	                #sFB_RightAngledTransfer_541(iUDT_Configuration := #iUDT_Configuration."541".RightAngledTransfer,
	                                             iUDT_LowerConveyorConfiguration := #iUDT_Configuration."540".Conveyor,
	                                             iUDT_UpperConveyorConfiguration := #iUDT_Configuration."541".Conveyor,
	                                             iUDT_PECConfiguration := #iUDT_Configuration."540".PEC,
	                                             ii_DestinationA := #si_540DestinationA,
	                                             ii_DestinationB := #si_540DestinationB,
	                                             ii_DestinationC := #si_540DestinationC,
	                                             ii_DestinationD := #si_540DestinationD,
	                                             ix_HardwareOk := #ix_HardwareOk,
	                                             ix_400vOk := #ix_400vOk,
	                                             ix_24vOk := #ix_24vOk,
	                                             ix_SafetyOk := #ix_SafetyOk,
	                                             ix_AirPressureOk := #ix_AirPressureOk,
	                                             ix_SectionIsDown := #ix_SectionIsDown541,
	                                             ix_SectionIsUp := #ix_SectionIsUp541,
	                                             ix_ConveyorAAuto := #iqUDT_WorkstationCommonStatus."530".AutoON,
	                                             ix_ConveyorBAuto := #iqUDT_WorkstationCommonStatus."550".AutoON,
	                                             ix_ConveyorCAuto := #iqUDT_WorkstationCommonStatus."670".AutoON,
	                                             ix_ConveyorDAuto := FALSE,
	                                             ix_PEC := #iUDT_MotorInput540.AllSensorPortInputs.LeftSensor,
	                                             ix_ExternalReceiveRequestA := NOT #iqUDT_WorkstationStatus."530".PEC_Eos.PEC AND NOT #sx_TransferOut380 AND NOT #sx_TransferOut390,
	                                             ix_ExternalReceiveRequestB := false,
	                                             ix_ExternalReceiveRequestC := #sFB_RightAngledTransfer_671.qx_ExternalSendRequestC,
	                                             ix_ExternalReceiveRequestD := false,
	                                             ix_PECInfeedA := #iqUDT_WorkstationStatus."530".PEC_Eos.PEC,
	                                             ix_PECInfeedC := #iqUDT_WorkstationStatus."670".PEC_Eos.PEC,
	                                             qUDT_HMIRATStatus => #iqUDT_WorkstationStatus."541".RightAngledTransfer,
	                                             qUDT_HMIConveyorStatus => #iqUDT_WorkstationStatus."540".Conveyor,
	                                             qUDT_HMIPECStatus => #iqUDT_WorkstationStatus."540".PEC_Eos,
	                                             qUDT_RATStatus => #iqUDT_WorkstationCommonStatus."541",
	                                             qUDT_ConveyorStatus => #iqUDT_WorkstationCommonStatus."540",
	                                             qx_PopupControl => #qx_PopupControl541,
	                                             iqUDT_EquipmentControl := #iqUDT_EquipmentControl,
	                                             iqUDT_RATCommand := #iqUDT_WorkstationCommands."541".RightAngledTransfer,
	                                             iqUDT_ConveyorCommand := #iqUDT_WorkstationCommands."540".Conveyor,
	                                             iqUDT_RATStatistics := #iqUDT_WorkstationStatistics."541".RightAngledTransfer,
	                                             iqUDT_ConveyorStatistics := #iqUDT_WorkstationStatistics."540".Conveyor,
	                                             iqUDT_PECStatistics := #iqUDT_WorkstationStatistics."540".PEC_Eos,
	                                             iqUDT_HandShakeConveyorA := #sUDT_Handshake_530,
	                                             iqUDT_HandShakeConveyorB := #sUDT_Handshake_540,
	                                             iqUDT_HandShakeConveyorC := #sUDT_HandshakeUp_671,
	                                             iqUDT_HandShakeConveyorD := #tUDT_dummyHandshake,
	                                             iqUDT_LowerConveyorInterface := #sUDT_Interface_540,
	                                             iqUDT_UpperConveyorInterface := #sUDT_Interface_541,
	                                             iqUDT_RATPositioning := #iqUDT_RATPositioning540,
	                                             iqUDT_BladeStopEoSInterface := #tUDT_DummyBladeStop,
	                                             iqUDT_BladeStopBoSInterface := #tUDT_DummyBladeStop);

	            END_REGION

	            REGION MCO
	                #sFB_MCOConveyLinxAixController_541(iUDT_AixConfig := #iUDT_Configuration."541".MCO_M01,
	                                                    iUDT_AixInputsModule := #iUDT_MotorInput540,
	                                                    ii_PositionSetpoint := #iqUDT_RATPositioning540.Upper.EndPosition,
	                                                    ix_24vOk := #ix_24vOk,
	                                                    ix_SimulationModeActive := "DB_Memory".Simulation,
	                                                    ii_MotorPositionId := 2,
	                                                    ix_StartPositioning := #iqUDT_RATPositioning540.Upper.Start,
	                                                    ix_ResetPosition := #iqUDT_RATPositioning540.Upper.ResetPosition,
	                                                    qUDT_HMIStatus => #iqUDT_WorkstationStatus."541".MCO_M01,
	                                                    qx_Positioned => #iqUDT_RATPositioning540.Upper.Done,
	                                                    iqUDT_AixOutputsModule := #qUDT_MotorOutput540,
	                                                    iqUDT_ConveyorInterface := #sUDT_Interface_541,
	                                                    iqUDT_MCOStatistics := #iqUDT_WorkstationStatistics."541".MCO_M01);
	            END_REGION

	        END_REGION

	        REGION 550

	            REGION Displacement

	                #sFB_Displacement550(#sUDT_Interface_550);

	            END_REGION

	            REGION Tracking

	                #sFB_Tracking_550(iUDT_ConveyorCommonConfiguration := #iUDT_Configuration."550".Conveyor.Common,
	                                  iqa_TrackingData := #sa_TrackingArray_550,
	                                  iqUDT_ConveyorInterface := #sUDT_Interface_550,
	                                  iqUDT_HandshakeUp := #sUDT_Handshake_540,
	                                  iqUDT_Handshake := #sUDT_Handshake_550);
	            END_REGION

	            REGION EOS

	                #sFB_PECUpdate_550(iUDT_PECUpdateConfiguration := #iUDT_Configuration."550".PEC_EoS,
	                                   iUDT_ConveyorCommonConfiguration := #iUDT_Configuration."550".Conveyor.Common,
	                                   ix_PEC := #iUDT_MotorInput550.AllSensorPortInputs.LeftSensor,
	                                   ix_TeachingMode := FALSE,
	                                   qUDT_Status => #iqUDT_WorkstationStatus."550".PEC_EoS,
	                                   qi_GINwrite => #ti_dummy,
	                                   qx_PECFiltered => #tx_dummy,
	                                   iqa_TrackingData := #sa_TrackingArray_550,
	                                   iqUDT_ConveyorInterface := #sUDT_Interface_550,
	                                   iqUDT_UnknownGINRange := #iqUDT_UnknownGINRange,
	                                   iqUDT_FifoHeader := "DB_FIFOLostGIN".Header,
	                                   iqa_FifoData := "DB_FIFOLostGIN".Data,
	                                   iqUDT_Statistics := #iqUDT_WorkstationStatistics."550".PEC_EoS);

	            END_REGION

	            REGION Conveyor
	                #sFB_Conveyor_550(iUDT_ConveyorConfiguration := #iUDT_Configuration."550".Conveyor,
	                                  idi_PECEoSDistance := #iUDT_Configuration."550".PEC_EoS.Distance,
	                                  idi_PECBoSDistance := 0,
	                                  ii_ExternalSpeed := 0,
	                                  ix_SafetyOk := #ix_SafetyOk,
	                                  ix_24vOk := #ix_24vOk,
	                                  ix_400vOk := #ix_400vOk,
	                                  ix_HardwareOk := #ix_HardwareOk,
	                                  ix_PECEoS := #iqUDT_WorkstationStatus."550".PEC_EoS.PEC,
	                                  ix_PECBoS := TRUE,
	                                  ix_ExternalRequestHold := false,
	                                  qUDT_HMIStatus => #iqUDT_WorkstationStatus."550".Conveyor,
	                                  qUDT_Status => #iqUDT_WorkstationCommonStatus."550",
	                                  iqUDT_EquipmentControl := #iqUDT_EquipmentControl,
	                                  iqUDT_ConveyorCommand := #iqUDT_WorkstationCommands."550".Conveyor,
	                                  iqUDT_ConveyorInterface := #sUDT_Interface_550,
	                                  iqUDT_HandShakeUp := #sUDT_Handshake_540,
	                                  iqUDT_HandShake := #sUDT_Handshake_550,
	                                  iqUDT_Statistics := #iqUDT_WorkstationStatistics."550".Conveyor);
	            END_REGION

	            REGION MCO
	                #sFB_MCOConveyLinxAixController_550(iUDT_AixConfig := #iUDT_Configuration."550".MCO_M01,
	                                                    iUDT_AixInputsModule := #iUDT_MotorInput550,
	                                                    ix_24vOk := #ix_24vOk,
	                                                    ix_SimulationModeActive := "DB_Memory".Simulation,
	                                                    ii_MotorPositionId := 1,
	                                                    qUDT_HMIStatus => #iqUDT_WorkstationStatus."550".MCO_M01,
	                                                    iqUDT_AixOutputsModule := #qUDT_MotorOutput550,
	                                                    iqUDT_ConveyorInterface := #sUDT_Interface_550,
	                                                    iqUDT_MCOStatistics := #iqUDT_WorkstationStatistics."550".MCO_M01);
	            END_REGION
	        END_REGION

	        REGION 560


	            REGION Displacement

	                #sFB_Displacement560(#sUDT_Interface_560);

	            END_REGION

	            REGION Conveyor
	                #sFB_Conveyor_560(iUDT_ConveyorConfiguration := #iUDT_Configuration."560".Conveyor,
	                                  idi_PECEoSDistance := 0,
	                                  idi_PECBoSDistance := 0,
	                                  ii_ExternalSpeed := 0,
	                                  ix_SafetyOk := #ix_SafetyOk,
	                                  ix_24vOk := #ix_24vOk,
	                                  ix_400vOk := #ix_400vOk,
	                                  ix_HardwareOk := #ix_HardwareOk,
	                                  ix_PECEoS := TRUE,
	                                  ix_PECBoS := TRUE,
	                                  ix_ExternalRequestHold := false,
	                                  qUDT_HMIStatus => #iqUDT_WorkstationStatus."560".Conveyor,
	                                  qUDT_Status => #iqUDT_WorkstationCommonStatus."560",
	                                  iqUDT_EquipmentControl := #iqUDT_EquipmentControl,
	                                  iqUDT_ConveyorCommand := #iqUDT_WorkstationCommands."560".Conveyor,
	                                  iqUDT_ConveyorInterface := #sUDT_Interface_560,
	                                  iqUDT_HandShakeUp := #sUDT_Handshake_550,
	                                  iqUDT_HandShake := #sUDT_Handshake_560,
	                                  iqUDT_Statistics := #iqUDT_WorkstationStatistics."560".Conveyor);
	            END_REGION

	            REGION VFD

	                #sFB_VfdNORDPPO4_560(iUDT_VFDConfig := #iUDT_Configuration."560".VFD,
	                                     iUDT_VFDInputs := #iUDT_MotorInput560,
	                                     iUDT_MotorData := #iUDT_MotorData560,
	                                     ix_24vOk := #ix_24vOk,
	                                     ix_400vOk := #ix_400vOk,
	                                     ix_QuickStopDisable := TRUE,
	                                     ix_SimulationModeActive := "DB_Memory".Simulation,
	                                     qUDT_HMIStatus => #iqUDT_WorkstationStatus."560".VFD,
	                                     qUDT_VFDOutputs => #qUDT_MotorOutput560,
	                                     iqUDT_ConveyorInterface := #sUDT_Interface_560,
	                                     iqUDT_VFDStatistics := #iqUDT_WorkstationStatistics."560".VFD,
	                                     iqx_StartCommissioning := #iqx_StartComissioning560);

	            END_REGION

	        END_REGION

	        REGION 570

	            REGION Displacement

	                #sFB_Displacement570(#sUDT_Interface_570);

	            END_REGION

	            REGION EoS

	                #sFB_PEC_570(ix_PEC := #iUDT_MotorInput570.AllSensorPortInputs.LeftSensor,
	                             iUDT_PECConfiguration := #iUDT_Configuration."570".PEC_EoS,
	                             qUDT_HMIStatus => #iqUDT_WorkstationStatus."570".PEC_EoS,
	                             iqUDT_ConveyorInterface := #sUDT_Interface_570,
	                             iqUDT_PECStatistics := #iqUDT_WorkstationStatistics."570".PEC_EoS);

	            END_REGION

	            REGION Conveyor
	                #sFB_Conveyor_570(iUDT_ConveyorConfiguration := #iUDT_Configuration."570".Conveyor,
	                                  idi_PECEoSDistance := #iUDT_Configuration."570".PEC_EoS.Distance,
	                                  idi_PECBoSDistance := 0,
	                                  ii_ExternalSpeed := 0,
	                                  ix_SafetyOk := #ix_SafetyOk,
	                                  ix_24vOk := #ix_24vOk,
	                                  ix_400vOk := #ix_400vOk,
	                                  ix_HardwareOk := #ix_HardwareOk,
	                                  ix_PECEoS := #iqUDT_WorkstationStatus."570".PEC_EoS.PEC,
	                                  ix_PECBoS := TRUE,
	                                  ix_ExternalRequestHold := false,
	                                  qUDT_HMIStatus => #iqUDT_WorkstationStatus."570".Conveyor,
	                                  qUDT_Status => #iqUDT_WorkstationCommonStatus."570",
	                                  iqUDT_EquipmentControl := #iqUDT_EquipmentControl,
	                                  iqUDT_ConveyorCommand := #iqUDT_WorkstationCommands."570".Conveyor,
	                                  iqUDT_ConveyorInterface := #sUDT_Interface_570,
	                                  iqUDT_HandShakeUp := #sUDT_Handshake_560,
	                                  iqUDT_HandShake := #sUDT_Handshake_570,
	                                  iqUDT_Statistics := #iqUDT_WorkstationStatistics."570".Conveyor);
	            END_REGION

	            REGION MCO
	                #sFB_MCOConveyLinxAixController_570(iUDT_AixConfig := #iUDT_Configuration."570".MCO_M01,
	                                                    iUDT_AixInputsModule := #iUDT_MotorInput570,
	                                                    ix_24vOk := #ix_24vOk,
	                                                    ix_SimulationModeActive := "DB_Memory".Simulation,
	                                                    ii_MotorPositionId := 1,
	                                                    qUDT_HMIStatus => #iqUDT_WorkstationStatus."570".MCO_M01,
	                                                    iqUDT_AixOutputsModule := #qUDT_MotorOutput570,
	                                                    iqUDT_ConveyorInterface := #sUDT_Interface_570,
	                                                    iqUDT_MCOStatistics := #iqUDT_WorkstationStatistics."570".MCO_M01);
	            END_REGION
	        END_REGION

	        REGION 580

	            REGION Displacement

	                #sFB_Displacement580(#sUDT_Interface_580);

	            END_REGION

	            REGION EoS

	                #sFB_PEC_580(ix_PEC := #iUDT_MotorInput570.AllSensorPortInputs.RightSensor,
	                             iUDT_PECConfiguration := #iUDT_Configuration."580".PEC_EoS,
	                             qUDT_HMIStatus => #iqUDT_WorkstationStatus."580".PEC_EoS,
	                             iqUDT_ConveyorInterface := #sUDT_Interface_580,
	                             iqUDT_PECStatistics := #iqUDT_WorkstationStatistics."580".PEC_EoS);

	            END_REGION

	            REGION Conveyor
	                #iqUDT_HandshakeDownstream580.RTR := #iqUDT_HandshakeDownstream580.RTR OR #iqUDT_WorkstationStatus."580".PEC_EoS.PEC;
	                #sFB_Conveyor_580(iUDT_ConveyorConfiguration := #iUDT_Configuration."580".Conveyor,
	                                  idi_PECEoSDistance := #iUDT_Configuration."580".PEC_EoS.Distance,
	                                  idi_PECBoSDistance := 0,
	                                  ii_ExternalSpeed := 0,
	                                  ix_SafetyOk := #ix_SafetyOk,
	                                  ix_24vOk := #ix_24vOk,
	                                  ix_400vOk := #ix_400vOk,
	                                  ix_HardwareOk := #ix_HardwareOk,
	                                  ix_PECEoS := #iqUDT_WorkstationStatus."580".PEC_EoS.PEC,
	                                  ix_PECBoS := TRUE,
	                                  ix_ExternalRequestHold := false,
	                                  qUDT_HMIStatus => #iqUDT_WorkstationStatus."580".Conveyor,
	                                  qUDT_Status => #iqUDT_WorkstationCommonStatus."580",
	                                  iqUDT_EquipmentControl := #iqUDT_EquipmentControl,
	                                  iqUDT_ConveyorCommand := #iqUDT_WorkstationCommands."580".Conveyor,
	                                  iqUDT_ConveyorInterface := #sUDT_Interface_580,
	                                  iqUDT_HandShakeUp := #sUDT_Handshake_570,
	                                  iqUDT_HandShake := #iqUDT_HandshakeDownstream580,
	                                  iqUDT_Statistics := #iqUDT_WorkstationStatistics."580".Conveyor);
	            END_REGION
	            REGION MCO
	                #sFB_MCOConveyLinxAixController_580(iUDT_AixConfig := #iUDT_Configuration."580".MCO_M01,
	                                                    iUDT_AixInputsModule := #iUDT_MotorInput570,
	                                                    ix_24vOk := #ix_24vOk,
	                                                    ix_SimulationModeActive := "DB_Memory".Simulation,
	                                                    ii_MotorPositionId := 2,
	                                                    qUDT_HMIStatus => #iqUDT_WorkstationStatus."580".MCO_M01,
	                                                    iqUDT_AixOutputsModule := #qUDT_MotorOutput570,
	                                                    iqUDT_ConveyorInterface := #sUDT_Interface_580,
	                                                    iqUDT_MCOStatistics := #iqUDT_WorkstationStatistics."580".MCO_M01);
	            END_REGION
	        END_REGION
	    END_REGION
	END_IF;


END_FUNCTION_BLOCK

FUNCTION_BLOCK "FB_NerakLift"
{ S7_Optimized_Access := 'TRUE' }
VERSION : 0.1
// ATTRIBUTES
// AUTO_NUMBER = True
// BLOCK_NUMBER = 250
// END_ATTRIBUTES
   VAR_INPUT
      iUDT_Configuration { ExternalAccessible := 'False'; ExternalVisible := 'False'; ExternalWritable := 'False'} : "UDT_NerakLiftConfiguration";   // Configuration structure
      idi_PECEoSDistance { ExternalAccessible := 'False'; ExternalVisible := 'False'; ExternalWritable := 'False'} : DInt;   // PEC distance from the end of lift
      ix_SafetyOK { ExternalAccessible := 'False'; ExternalVisible := 'False'; ExternalWritable := 'False'} : Bool;   // TRUE when safety is ok
      ix_24VOk { ExternalAccessible := 'False'; ExternalVisible := 'False'; ExternalWritable := 'False'} : Bool;   // TRUE when 24V supply is ok
      ix_400VOk { ExternalAccessible := 'False'; ExternalVisible := 'False'; ExternalWritable := 'False'} : Bool;   // TRUE when 400V supply is ok
      ix_HardwareOk { ExternalAccessible := 'False'; ExternalVisible := 'False'; ExternalWritable := 'False'} : Bool;   // TRUE when hardware is ok
      iudt_IOIn { ExternalAccessible := 'False'; ExternalVisible := 'False'; ExternalWritable := 'False'} : "UDT_NerakLiftPI";   // Structure of inputs from IO Panel
   END_VAR

   VAR_OUTPUT
      qUDT_HMIStatus { ExternalAccessible := 'False'; ExternalVisible := 'False'; ExternalWritable := 'False'} : "UDT_NerakLiftStatus";   // HMI status structure
      qudt_IOOut { ExternalAccessible := 'False'; ExternalVisible := 'False'; ExternalWritable := 'False'} : "UDT_NerakLiftPO";   // Structure of outputs from IO Panel
      qx_Fault { ExternalAccessible := 'False'; ExternalVisible := 'False'; ExternalWritable := 'False'} : Bool;   // Fault active
      qx_Ready { ExternalAccessible := 'False'; ExternalVisible := 'False'; ExternalWritable := 'False'} : Bool;   // Machine ready
      qx_ExternalDieback { ExternalAccessible := 'False'; ExternalVisible := 'False'; ExternalWritable := 'False'} : Bool;   // Send external dieback to downstream conveyor
   END_VAR

   VAR_IN_OUT
      iqUDT_CommonStatus : "UDT_CommonStatus";   // Common status structure
      iqUDT_EquipmentControl : "UDT_EquipmentControl";   // Equipment control structure
      iqUDT_HandshakeUp : "UDT_ConveyorHandshake";   // Upstream handshake structure
      iqUDT_Handshake : "UDT_ConveyorHandshake";   // Downstream handshake structure
      iqUDT_Interface : "UDT_ConveyorInterface";   // Interface structure
      iqUDT_ConveyorCommand : "UDT_ConveyorCommand";   // HMI commands structure
      iqUDT_Statistics : "UDT_NerakLiftStatistics";   // Statistics structure
   END_VAR

   VAR
      sUDT_HMIStatus { ExternalAccessible := 'False'; ExternalVisible := 'False'; ExternalWritable := 'False'; S7_SetPoint := 'False'} : "UDT_NerakLiftStatus";   // HMI status structure
      sUDT_ConveyorConfiguration { ExternalAccessible := 'False'; ExternalVisible := 'False'; ExternalWritable := 'False'; S7_SetPoint := 'False'} : "UDT_ConveyorConfiguration" := (((), 0), (), (), (), 0, 200, (), (), FALSE);   // Conveyor configuration structure
      sFB_ConveyorControl { ExternalAccessible := 'False'; ExternalVisible := 'False'; ExternalWritable := 'False'; S7_SetPoint := 'False'} : "FB_Conveyor";   // Conveyor instance
      sFB_TimerOnOffDelay_B2Treshold { ExternalAccessible := 'False'; ExternalVisible := 'False'; ExternalWritable := 'False'; S7_SetPoint := 'False'} : "FB_TimerOnOffDelay";   // B2 on off delay
      sFB_TimerOnOffDelay_B3Treshold { ExternalAccessible := 'False'; ExternalVisible := 'False'; ExternalWritable := 'False'; S7_SetPoint := 'False'} : "FB_TimerOnOffDelay";   // B3 on off delay
      sFB_TimerOnOffDelay_B4Treshold { ExternalAccessible := 'False'; ExternalVisible := 'False'; ExternalWritable := 'False'; S7_SetPoint := 'False'} : "FB_TimerOnOffDelay";   // B4 on off delay
      sFB_TimerOnOffDelay_B5Treshold { ExternalAccessible := 'False'; ExternalVisible := 'False'; ExternalWritable := 'False'; S7_SetPoint := 'False'} : "FB_TimerOnOffDelay";   // B5 on off delay
      sFB_TimerOnOffDelay_B10Treshold { ExternalAccessible := 'False'; ExternalVisible := 'False'; ExternalWritable := 'False'; S7_SetPoint := 'False'} : "FB_TimerOnOffDelay";   // B10 on off delay
      sFB_TimerOnOffDelay_B11Treshold { ExternalAccessible := 'False'; ExternalVisible := 'False'; ExternalWritable := 'False'; S7_SetPoint := 'False'} : "FB_TimerOnOffDelay";   // B11 on off delay
      sR_TRIG_ProductFellDown {InstructionName := 'R_TRIG'; LibVersion := '1.0'; ExternalAccessible := 'False'; ExternalVisible := 'False'; ExternalWritable := 'False'; S7_SetPoint := 'False'} : R_TRIG;   // R_TRIG Product fell down for statistics
      sR_TRIG_CollisionDetected {InstructionName := 'R_TRIG'; LibVersion := '1.0'; ExternalAccessible := 'False'; ExternalVisible := 'False'; ExternalWritable := 'False'; S7_SetPoint := 'False'} : R_TRIG;   // R_TRIG collision detected for statistics
      sx_B2Filtered { ExternalAccessible := 'False'; ExternalVisible := 'False'; ExternalWritable := 'False'} : Bool;   // B2 sensor filtered
      sx_B3Filtered { ExternalAccessible := 'False'; ExternalVisible := 'False'; ExternalWritable := 'False'} : Bool;   // Cumulative B3 sensors filtered
      sx_B4Filtered { ExternalAccessible := 'False'; ExternalVisible := 'False'; ExternalWritable := 'False'} : Bool;   // B4 sensor filtered
      sx_B5Filtered { ExternalAccessible := 'False'; ExternalVisible := 'False'; ExternalWritable := 'False'} : Bool;   // B5 sensor filtered
      sx_B10Filtered { ExternalAccessible := 'False'; ExternalVisible := 'False'; ExternalWritable := 'False'} : Bool;   // B10 sensor filtered
      sx_B11Filtered { ExternalAccessible := 'False'; ExternalVisible := 'False'; ExternalWritable := 'False'} : Bool;   // B11 sensor filtered
   END_VAR

   VAR_TEMP
      tUDT_Statistics : "UDT_ConveyorStatistics";   // Temporary conveyor statistics structure
      tUDT_ConveyorHMIStatus : "UDT_ConveyorStatus";   // Temporary conveyor status structure
      tx_ExternalDieback : Bool;   // Upstream dieback control
      tx_Hold : Bool;   // Hold bit
      tx_GlobalResetMemory : Bool;   // Memory for global reset
   END_VAR


BEGIN
	(*
	----------------------------------------------------------------------------------------

	Version history:
	Date        | Version   | Author        | Remark
	----------------------------------------------------------------------------------------
	20/02/2024  | 1.0       | K.Pokorski    | First release TIA 17
	28/03/2024  | 1.1       | K. Pokorski   | Modifications after lift test
	16/08/2024  | 2.0       | J.Majer       | Block Interface IO changed to UDT type
	*)

	REGION 1 - Edge detection

	    #sR_TRIG_ProductFellDown(CLK := #sUDT_HMIStatus.Specific.ProductFellDown);

	    #sR_TRIG_CollisionDetected(CLK := #sUDT_HMIStatus.Specific.CollisionDetected);

	END_REGION

	REGION 2 - Filtering

	    #sFB_TimerOnOffDelay_B2Treshold(iudi_OnDelayTime := #iUDT_Configuration.CollisionSensorDelayOn,
	                                    iudi_OffDelayTime := #iUDT_Configuration.CollisionSensorDelayOff,
	                                    ix_SignalToDelay := #iudt_IOIn.ix_B2_CollisionControl,
	                                    qx_DelayedSignal => #sx_B2Filtered);

	    #sFB_TimerOnOffDelay_B3Treshold(iudi_OnDelayTime := #iUDT_Configuration.FallingThroughSensorDelayOn,
	                                    iudi_OffDelayTime := #iUDT_Configuration.FallingThroughSensorDelayOff,
	                                    ix_SignalToDelay := #iudt_IOIn."ix_B3.1FallingThrought" AND #iudt_IOIn."ix_B3.2FallingThrought" AND #iudt_IOIn."ix_B3.3FallingThrought",
	                                    qx_DelayedSignal => #sx_B3Filtered);

	    #sFB_TimerOnOffDelay_B4Treshold(iudi_OnDelayTime := #iUDT_Configuration.TailbackControlFrontSensorDelayOn,
	                                    iudi_OffDelayTime := #iUDT_Configuration.TailbackControlFrontSensorDelayOff,
	                                    ix_SignalToDelay := #iudt_IOIn.ix_B4TailbackControlFront,
	                                    qx_DelayedSignal => #sx_B4Filtered);

	    #sFB_TimerOnOffDelay_B5Treshold(iudi_OnDelayTime := #iUDT_Configuration.TailbackControlRearSensorDelayOn,
	                                    iudi_OffDelayTime := #iUDT_Configuration.TailbackControlRearSensorDelayOff,
	                                    ix_SignalToDelay := #iudt_IOIn.ix_B5TailbackControlBack,
	                                    qx_DelayedSignal => #sx_B5Filtered);

	    #sFB_TimerOnOffDelay_B10Treshold(iudi_OnDelayTime := #iUDT_Configuration.PlatformPositionSensorDelayOn,
	                                     iudi_OffDelayTime := #iUDT_Configuration.PlatformPositionSensorDelayOff,
	                                     ix_SignalToDelay := #iudt_IOIn.ix_B10_PlatforninPosition,
	                                     qx_DelayedSignal => #sx_B10Filtered);

	    #sFB_TimerOnOffDelay_B11Treshold(iudi_OnDelayTime := #iUDT_Configuration.CollisionSensorDelayOn,
	                                     iudi_OffDelayTime := #iUDT_Configuration.CollisionSensorDelayOff,
	                                     ix_SignalToDelay := #iudt_IOIn.ix_B11ColisionControl,
	                                     qx_DelayedSignal => #sx_B11Filtered);

	END_REGION

	REGION 3 - Errors

	    IF #iqUDT_EquipmentControl.Command.Reset OR #iudt_IOIn.ix_FaultReset
	    THEN
	        #sUDT_HMIStatus.Specific.CollisionDetected := FALSE;
	        #sUDT_HMIStatus.Specific.ProductFellDown := FALSE;
	    END_IF;

	    IF NOT #sx_B2Filtered AND #sx_B11Filtered AND #iUDT_Configuration.Mode = 1
	        OR NOT #sx_B2Filtered AND #iUDT_Configuration.Mode = 2
	    THEN
	        #sUDT_HMIStatus.Specific.CollisionDetected := TRUE;
	    END_IF;

	    IF NOT #sx_B3Filtered
	    THEN
	        #sUDT_HMIStatus.Specific.ProductFellDown := TRUE;
	    END_IF;

	    IF #sUDT_HMIStatus.Specific.CollisionDetected
	        OR #sUDT_HMIStatus.Specific.ProductFellDown THEN
	        #iqUDT_Interface.InternalErrorPEC := TRUE;
	    END_IF;

	END_REGION

	REGION 4 - Conveyor control

	    REGION 4.1 - Conveyor configuration

	        #sUDT_ConveyorConfiguration.Common.Length := #iUDT_Configuration.Length;
	        #sUDT_ConveyorConfiguration.Forward_Direction.EnergySaveLenght := #iUDT_Configuration.EnergySaveLength;
	        #sUDT_ConveyorConfiguration.Forward_Direction.PEC_EoSDistanceOffset := #iUDT_Configuration.PEC_EoSDistanceOffset;
	        #sUDT_ConveyorConfiguration.Forward_Direction.FirstConveyorToStart := #iUDT_Configuration.FirstConveyorToStart;
	        #sUDT_ConveyorConfiguration.CascadeTimeOnDelay := #iUDT_Configuration.CascadeTimeOnDelay;
	        #sUDT_ConveyorConfiguration.SpeedSetpointNominal := #iUDT_Configuration.SpeedSetpointNominal;
	        #sUDT_ConveyorConfiguration.Energy := #iUDT_Configuration.Energy;

	    END_REGION

	    REGION 4.2 - Tailback control

	        #tx_Hold := NOT #sx_B4Filtered AND NOT #sx_B5Filtered;

	    END_REGION

	    REGION 4.3 - Conveyor block call

	        #tx_GlobalResetMemory := #iqUDT_EquipmentControl.Command.Reset;
	        #iqUDT_EquipmentControl.Command.Reset := #iqUDT_EquipmentControl.Command.Reset OR #iudt_IOIn.ix_FaultReset;

	        #iqUDT_ConveyorCommand.ManualMode := #iudt_IOIn.ix_ManualMode;
	        #iqUDT_ConveyorCommand.ManualStartStop := FALSE;
	        #iqUDT_ConveyorCommand.ManualJog := #iudt_IOIn.ix_ManualUp OR #iudt_IOIn.ix_ManualDown;

	        #iqUDT_ConveyorCommand.Reverse :=
	        (#iUDT_Configuration.Mode = 1 AND #iudt_IOIn.ix_ManualUp)
	        OR (#iUDT_Configuration.Mode = 2 AND #iudt_IOIn.ix_ManualDown);

	        #sFB_ConveyorControl(iUDT_ConveyorConfiguration := #sUDT_ConveyorConfiguration,
	                             idi_PECEoSDistance := #idi_PECEoSDistance,
	                             idi_PECBoSDistance := 0,
	                             ii_ExternalSpeed := 0,
	                             ix_SafetyOk := #ix_SafetyOK,
	                             ix_24vOk := #ix_24VOk,
	                             ix_400vOk := #ix_400VOk,
	                             ix_HardwareOk := #ix_HardwareOk,
	                             ix_PECEoS := #sx_B5Filtered,
	                             ix_PECBoS := TRUE,
	                             ix_ReverseDirection := FALSE,
	                             ix_ExternalRequestDieBack := FALSE,
	                             ix_ExternalRequestHold := #tx_Hold,
	                             ix_ResetEnergySave := FALSE,
	                             qUDT_HMIStatus => #tUDT_ConveyorHMIStatus,
	                             qUDT_Status => #iqUDT_CommonStatus,
	                             iqUDT_EquipmentControl := #iqUDT_EquipmentControl,
	                             iqUDT_ConveyorCommand := #iqUDT_ConveyorCommand,
	                             iqUDT_ConveyorInterface := #iqUDT_Interface,
	                             iqUDT_HandShakeUp := #iqUDT_HandshakeUp,
	                             iqUDT_HandShake := #iqUDT_Handshake,
	                             iqUDT_Statistics := #tUDT_Statistics);

	        IF #iqUDT_CommonStatus.ManualRun
	            AND #iqUDT_Interface.SpeedSetpoint > 200
	        THEN
	            #iqUDT_Interface.SpeedSetpoint := 200;
	        END_IF;

	        #iqUDT_EquipmentControl.Command.Reset := #tx_GlobalResetMemory;
	        #tx_ExternalDieback := TRUE;
	        IF #sx_B10Filtered THEN
	            #tx_ExternalDieback := false;
	        END_IF;

	    END_REGION

	END_REGION

	REGION 5 - Status

	    #sUDT_HMIStatus.Status := #tUDT_ConveyorHMIStatus.Status;
	    #qUDT_HMIStatus := #sUDT_HMIStatus;

	END_REGION

	REGION 6 - Statistics

	    REGION 6.1 - Conveyor statistics mapping

	        #iqUDT_Statistics.EnergySave := #tUDT_Statistics.EnergySave;
	        #iqUDT_Statistics.ConveyorStop := #tUDT_Statistics.ConveyorStop;
	        #iqUDT_Statistics.ConveyorDown := #tUDT_Statistics.ConveyorDown;
	        #iqUDT_Statistics.ConveyorUp := #tUDT_Statistics.ConveyorUp;

	    END_REGION

	    REGION 6.2 - Collision detected time

	        IF #sUDT_HMIStatus.Specific.CollisionDetected OR #iqUDT_EquipmentControl.Command.ResetData  // Reset statistics
	        THEN

	            "FC_Statistics"(ix_Reset := #iqUDT_EquipmentControl.Command.ResetData,          // Reset statistics input
	                            ix_Activate := #sUDT_HMIStatus.Specific.CollisionDetected,         // Activate statistics functions input
	                            ix_RTrigActivate := #sR_TRIG_CollisionDetected.Q,                       // Statistics active trigger
	                            iqUDT_Statistics := #iqUDT_Statistics.CollisionDetected);               // Statistics values output

	        END_IF;

	    END_REGION

	    REGION 6.3 - Collision detected time

	        IF #sUDT_HMIStatus.Specific.ProductFellDown OR #iqUDT_EquipmentControl.Command.ResetData  // Reset statistics
	        THEN

	            "FC_Statistics"(ix_Reset := #iqUDT_EquipmentControl.Command.ResetData,          // Reset statistics input
	                            ix_Activate := #sUDT_HMIStatus.Specific.ProductFellDown,         // Activate statistics functions input
	                            ix_RTrigActivate := #sR_TRIG_ProductFellDown.Q,                       // Statistics active trigger
	                            iqUDT_Statistics := #iqUDT_Statistics.ProductFellDown);               // Statistics values output

	        END_IF;

	    END_REGION

	END_REGION

	REGION 7 - Outputs

	    #qx_Fault := #iqUDT_CommonStatus.Error;
	    #qx_Ready := NOT #iqUDT_CommonStatus.Error;
	    #qx_ExternalDieback := #tx_ExternalDieback;

	END_REGION
END_FUNCTION_BLOCK

FUNCTION_BLOCK "FB_TGWLift"
{ S7_Optimized_Access := 'TRUE' }
VERSION : 0.1
// ATTRIBUTES
// AUTO_NUMBER = True
// BLOCK_NUMBER = 272
// END_ATTRIBUTES
   VAR_INPUT
      iUDT_TGWLiftConfiguration { ExternalAccessible := 'False'; ExternalVisible := 'False'; ExternalWritable := 'False'} : "UDT_TGWLiftConfiguration";   // Lift configuration structure
      iUDT_010MotorInput { ExternalAccessible := 'False'; ExternalVisible := 'False'; ExternalWritable := 'False'} : "UDT_VfdSEWSpeedPI";   // 010 SEW inputs structure
      iUDT_020MotorInput { ExternalAccessible := 'False'; ExternalVisible := 'False'; ExternalWritable := 'False'} : "UDT_VfdSEWPositioningPI";   // 020 SEW Positioning structure
      is_ET200spPNDeviceName { ExternalAccessible := 'False'; ExternalVisible := 'False'; ExternalWritable := 'False'} : String;   // Name of ET200
      ix_010EoS { ExternalAccessible := 'False'; ExternalVisible := 'False'; ExternalWritable := 'False'} : Bool;   // End of the section - Lift conveyor
      ix_010BoS { ExternalAccessible := 'False'; ExternalVisible := 'False'; ExternalWritable := 'False'} : Bool;   // Begining of the section - Lift conveyor
      ix_010PECMiddle { ExternalAccessible := 'False'; ExternalVisible := 'False'; ExternalWritable := 'False'} : Bool;   // Middle of the section - Lift conveyor
      ix_010PECGapBegin { ExternalAccessible := 'False'; ExternalVisible := 'False'; ExternalWritable := 'False'} : Bool;   // Gap Check Beginning
      ix_010PECGapEnd { ExternalAccessible := 'False'; ExternalVisible := 'False'; ExternalWritable := 'False'} : Bool;   // Gap Check End
      iUDT_LiftPI { ExternalAccessible := 'False'; ExternalVisible := 'False'; ExternalWritable := 'False'} : "UDT_TGWLiftPI";   // Reading inputs from the input card
      ix_24vOk { ExternalAccessible := 'False'; ExternalVisible := 'False'; ExternalWritable := 'False'} : Bool;   // TRUE when 24VDC is healthy
      ix_400vOk { ExternalAccessible := 'False'; ExternalVisible := 'False'; ExternalWritable := 'False'} : Bool;   // TRUE when 400VAC is healthy
      ix_SafetyOk { ExternalAccessible := 'False'; ExternalVisible := 'False'; ExternalWritable := 'False'} : Bool;   // TRUE when safety is ok
      ix_HardwareOk { ExternalAccessible := 'False'; ExternalVisible := 'False'; ExternalWritable := 'False'} : Bool;   // TRUE when hardware is ok
      ix_MaintSupport1 { ExternalAccessible := 'False'; ExternalVisible := 'False'; ExternalWritable := 'False'} : Bool;   // Lift supporting maintenance platform 1 retracted
      ix_MaintSupport2 { ExternalAccessible := 'False'; ExternalVisible := 'False'; ExternalWritable := 'False'} : Bool;   // Lift supporting maintenance platform 2 retracted
      ix_KeySwitchStop { ExternalAccessible := 'False'; ExternalVisible := 'False'; ExternalWritable := 'False'} : Bool;   // Key switch stop
      ix_LimitSwitchUp { ExternalAccessible := 'False'; ExternalVisible := 'False'; ExternalWritable := 'False'} : Bool;   // Limit switch up
      ix_LimitSwitchDown { ExternalAccessible := 'False'; ExternalVisible := 'False'; ExternalWritable := 'False'} : Bool;   // Limit switch down
   END_VAR

   VAR_OUTPUT
      qUDT_010MotorOutput { ExternalAccessible := 'False'; ExternalVisible := 'False'; ExternalWritable := 'False'} : "UDT_VfdSEWSpeedPO";   // 010 SEW outputs structure
      qUDT_020MotorOutput { ExternalAccessible := 'False'; ExternalVisible := 'False'; ExternalWritable := 'False'} : "UDT_VfdSEWPositioningPO";   // 020 SEW positioning outputs structure
      qUDT_LiftPO { ExternalAccessible := 'False'; ExternalVisible := 'False'; ExternalWritable := 'False'} : "UDT_TGWLiftPO";   // writing outputs to the output card
   END_VAR

   VAR_IN_OUT
      iqUDT_EquipmentControl : "UDT_EquipmentControl";   // Equipment control structure
      iqUDT_TGWLiftHMICommands : "UDT_TGWLiftHmiCommands";   // HMI commands structure for lift
      iqUDT_TGWLiftCommonStatus : "UDT_TGWLiftCommonStatus";   // Common status structure for 010 conveyor
      iqUDT_TGWLiftStatus : "UDT_TGWLiftStatus";   // Status TGW Lift structure
      iqUDT_TGWLiftStatistics : "UDT_TGWLiftStatistics";   // Statistics TGW Lift structure
      iqUDT_InfeedFullDownHMICommands : "UDT_ConveyorCommand";   // HMI commands structure for lower infeed conveyor
      iqUDT_OutfeedEmptyDownHMICommands : "UDT_ConveyorCommand";   // HMI commands structure for lower outfeed conveyor
      iqUDT_InfeedEmptyUpHMICommands : "UDT_ConveyorCommand";   // HMI commands structure for upper infeed conveyor
      iqUDT_OutfeedFullUpHMICommands : "UDT_ConveyorCommand";   // HMI commands structure for upper outfeed conveyor
      iqUDT_InfeedFullDownCommonStatus : "UDT_CommonStatus";   // Common status structure for full infeed conveyor
      iqUDT_OutfeedEmptyDownCommonStatus : "UDT_CommonStatus";   // Common status structure for empty outfeed conveyor
      iqUDT_InfeedEmptyUpCommonStatus : "UDT_CommonStatus";   // Common status structure for empty infeed
      iqUDT_OutfeedFullupCommonStatus : "UDT_CommonStatus";   // Common status structure for full outfeed conveyor
      iqUDT_InfeedFullDownHandShake : "UDT_ConveyorHandshake";   // Handshake structure for full infeed conveyor
      iqUDT_OutfeedEmptyDownHandShake : "UDT_ConveyorHandshake";   // Handshake structure for empty outfeed conveyor
      iqUDT_InfeedEmptyUpHandShake : "UDT_ConveyorHandshake";   // Handshake structure for empty infeed conveyor
      iqUDT_OutfeedFullUpHandShake : "UDT_ConveyorHandshake";   // Handshake structure for full outfeed conveyor
      iqUDT_OutfeedEmptyDownHandshakeUpstream : "UDT_ConveyorHandshake";   // HandshakeUp structure for empty outfeed conveyor
      iqUDT_OutfeedFullUpHandshakeUpstream : "UDT_ConveyorHandshake";   // HandshakeUp structure for full outfeed conveyor
   END_VAR

   VAR
      sUDT_020VSUInterface { ExternalAccessible := 'False'; ExternalVisible := 'False'; ExternalWritable := 'False'; S7_SetPoint := 'False'} : "UDT_VSUInterface";   // Interface structure for lift 020
      sUDT_010ConveyorInterface { ExternalAccessible := 'False'; ExternalVisible := 'False'; ExternalWritable := 'False'; S7_SetPoint := 'False'} : "UDT_ConveyorInterface";   // Interface structure for conveyor 010
      sFB_010Displacement { ExternalAccessible := 'False'; ExternalVisible := 'False'; ExternalWritable := 'False'; S7_SetPoint := 'False'} : "FB_Displacement";   // Displacement calculation for 010 conveyor
      sFB_010PECEoS { ExternalAccessible := 'False'; ExternalVisible := 'False'; ExternalWritable := 'False'; S7_SetPoint := 'False'} : "FB_PEC";   // Photoeye EoS handling for 010 conveyor
      sFB_010PECBoS { ExternalAccessible := 'False'; ExternalVisible := 'False'; ExternalWritable := 'False'; S7_SetPoint := 'False'} : "FB_PEC";   // Photoeye BoS handling for 010 conveyor
      sFB_LiftManualControl { ExternalAccessible := 'False'; ExternalVisible := 'False'; ExternalWritable := 'False'; S7_SetPoint := 'False'} : "FB_LiftManualControl";   // Function block to control lift, infeeds and outfeeds manually
      sFB_010Conveyor { ExternalAccessible := 'False'; ExternalVisible := 'False'; ExternalWritable := 'False'; S7_SetPoint := 'False'} : "FB_Conveyor";   // Function block to control the 010 conveyor
      sFB_010VfdSEWMOVICSpeed { ExternalAccessible := 'False'; ExternalVisible := 'False'; ExternalWritable := 'False'; S7_SetPoint := 'False'} : "FB_VfdSEWMOVI-CSpeed";   // Function to interface with SEW-MoviCSpeed for  010
      sFB_020VfdSEWMOVICPositioning { ExternalAccessible := 'False'; ExternalVisible := 'False'; ExternalWritable := 'False'; S7_SetPoint := 'False'} : "FB_VfdSEWMOVI-CPositioning";   // Function to interface with SEW-MoviCPositioning for  020
      sFB_020RIOVSU { ExternalAccessible := 'False'; ExternalVisible := 'False'; ExternalWritable := 'False'; S7_SetPoint := 'False'} : "FB_RIOVSU";   // Function block of RIO VSU
      sFB_020Lift { ExternalAccessible := 'False'; ExternalVisible := 'False'; ExternalWritable := 'False'; S7_SetPoint := 'False'} : "FB_Lift";   // Function block for lift control
      sFB_020VSULift { ExternalAccessible := 'False'; ExternalVisible := 'False'; ExternalWritable := 'False'; S7_SetPoint := 'False'} : "FB_VSULift";   // Funcion block of VSU Lift
      sUDT_010HandshakeUp { ExternalAccessible := 'False'; ExternalVisible := 'False'; ExternalWritable := 'False'; S7_SetPoint := 'False'} : "UDT_ConveyorHandshake";   // HandshakeUp structure for 010
      sUDT_010Handshake { ExternalAccessible := 'False'; ExternalVisible := 'False'; ExternalWritable := 'False'; S7_SetPoint := 'False'} : "UDT_ConveyorHandshake";   // Handshake structure for 010
   END_VAR

   VAR_TEMP
      tx_LiftConveyorDirection : Bool;   // Direction of lift conveyor
   END_VAR

   VAR CONSTANT
      ci_LiftUp : Int := 2;   // Constant for indicating Lift up position
      ci_LiftDown : Int := 1;   // Constant for indicating Lift down position
   END_VAR


BEGIN
	(*
	----------------------------------------------------------------------------------------

	Version history:
	Date        | Version   | Author        | Remark
	----------------------------------------------------------------------------------------
	06/08/2024  | 1.0       | R. Pieczonka  | Initial version
	12/08/2024  | 1.1       | R. Pieczonka  | Changing the block interface from struct to UDT types
	            |           | J.Majer       | Changing input & Outputs to UDT type
	*)


	REGION LFTxx-010
	    // Autostore picking station lift conveyor
	    // Function variant: TV11

	    REGION Displacement
	        #sFB_010Displacement(#sUDT_010ConveyorInterface);

	    END_REGION

	    REGION EOS
	        #sFB_010PECEoS(ix_PEC := #ix_010EoS,
	                       iUDT_PECConfiguration := #iUDT_TGWLiftConfiguration."010".PEC_EoS,
	                       qUDT_HMIStatus => #iqUDT_TGWLiftStatus."010".PEC_EoS,
	                       iqUDT_ConveyorInterface := #sUDT_010ConveyorInterface,
	                       iqUDT_PECStatistics := #iqUDT_TGWLiftStatistics."010".PEC_EoS);

	    END_REGION

	    REGION BOS
	        #sFB_010PECBoS(ix_PEC := #ix_010BoS,
	                       iUDT_PECConfiguration := #iUDT_TGWLiftConfiguration."010".PEC_BoS,
	                       qUDT_HMIStatus => #iqUDT_TGWLiftStatus."010".PEC_BoS,
	                       iqUDT_ConveyorInterface := #sUDT_010ConveyorInterface,
	                       iqUDT_PECStatistics := #iqUDT_TGWLiftStatistics."010".PEC_BoS);

	    END_REGION

	    REGION Manual Control
	        #sFB_LiftManualControl(ix_ManualMode := #iUDT_LiftPI.ix_ManualMode,                                     // Manual mode
	                               ix_AutoMode := #iUDT_LiftPI.ix_AutoMode,                                         // Auto mode
	                               ix_UpPosition := #sUDT_020VSUInterface.PositionActual = #ci_LiftUp,
	                               ix_DownPosition := #sUDT_020VSUInterface.PositionActual = #ci_LiftDown,
	                               ix_LiftConveyorRight := #iUDT_LiftPI.ix_LiftConveyorFwd,
	                               ix_LiftConveyorLeft := #iUDT_LiftPI.ix_LiftConveyorRvs,
	                               ix_InfeedConveyor := #iUDT_LiftPI.ix_InfeedConveyor,
	                               ix_OutfeedConveyor := #iUDT_LiftPI.ix_OutfeedConveyor,
	                               iqUDT_LiftConveyorCommand := #iqUDT_TGWLiftHMICommands."010".Conveyor,
	                               iqUDT_LowerInfeedConveyorCommand := #iqUDT_InfeedFullDownHMICommands,
	                               iqUDT_LowerOutfeedConveyorCommand := #iqUDT_OutfeedEmptyDownHMICommands,
	                               iqUDT_UpperInfeedConveyorCommand := #iqUDT_InfeedEmptyUpHMICommands,
	                               iqUDT_UpperOutfeedConveyorCommand := #iqUDT_OutfeedFullUpHMICommands);

	    END_REGION

	    REGION Conveyor


	        #sFB_010Conveyor(iUDT_ConveyorConfiguration := #iUDT_TGWLiftConfiguration."010".Conveyor,
	                         idi_PECEoSDistance := #iUDT_TGWLiftConfiguration."010".PEC_EoS.Distance,
	                         idi_PECBoSDistance := #iUDT_TGWLiftConfiguration."010".PEC_BoS.Distance,
	                         ii_ExternalSpeed := 0,
	                         ix_SafetyOk := #ix_SafetyOk,
	                         ix_24vOk := #ix_24vOk AND #iUDT_LiftPI.ix_F1400ok,
	                         ix_400vOk := #ix_400vOk AND #iUDT_LiftPI.ix_F1002ok,
	                         ix_HardwareOk := #ix_HardwareOk,
	                         ix_PECEoS := #iqUDT_TGWLiftStatus."010".PEC_EoS.PEC,
	                         ix_PECBoS := #iqUDT_TGWLiftStatus."010".PEC_BoS.PEC,
	                         ix_ReverseDirection := #sFB_020Lift.qx_LiftConveyorDirection,
	                         ix_ExternalRequestHold := NOT (#sUDT_020VSUInterface.PositionActual = #ci_LiftUp OR #sUDT_020VSUInterface.PositionActual = #ci_LiftDown),
	                         qUDT_HMIStatus => #iqUDT_TGWLiftStatus."010".Conveyor,
	                         qUDT_Status => #iqUDT_TGWLiftCommonStatus."010",
	                         iqUDT_EquipmentControl := #iqUDT_EquipmentControl,
	                         iqUDT_ConveyorCommand := #iqUDT_TGWLiftHMICommands."010".Conveyor,
	                         iqUDT_ConveyorInterface := #sUDT_010ConveyorInterface,
	                         iqUDT_HandShakeUp := #sUDT_010HandshakeUp,
	                         iqUDT_HandShake := #sUDT_010Handshake,
	                         iqUDT_Statistics := #iqUDT_TGWLiftStatistics."010".Conveyor);



	    END_REGION

	    REGION VFD

	        #"sFB_010VfdSEWMOVICSpeed"(iUDT_VfdConfig := #iUDT_TGWLiftConfiguration."010".VFD,
	                                   iUDT_VfdInputs := #iUDT_010MotorInput,
	                                   ix_PowerOK := TRUE,
	                                   ix_SimulationModeActive := FALSE,
	                                   ix_QuickStopDisable := TRUE,
	                                   qUDT_HMIStatus => #iqUDT_TGWLiftStatus."010".VFD,
	                                   qUDT_VfdOutputs => #qUDT_010MotorOutput,
	                                   iqUDT_ConveyorInterface := #sUDT_010ConveyorInterface,
	                                   iqUDT_VfdStatistics := #iqUDT_TGWLiftStatistics."010".VFD);

	    END_REGION

	END_REGION

	REGION LFTxx-020
	    // Autostore picking station lift positioning
	    // Function variant: VL11

	    REGION VSU RIO
	        #sFB_020RIOVSU(is_ET200spPNDeviceName := #is_ET200spPNDeviceName,
	                       ix_400VintOk := #ix_400vOk AND #iUDT_LiftPI.ix_F1002ok,
	                       ix_400VextOk := #iUDT_LiftPI.ix_MainSwitchCabinetOn AND #ix_400vOk AND #iUDT_LiftPI.ix_F1002ok,
	                       ix_BrakeSupplyOk := #ix_400vOk AND #iUDT_LiftPI.ix_F1002ok,
	                       ix_ThermalBrake := #iUDT_LiftPI.ix_OverTempBrakeRes,
	                       ix_24VOk := #ix_24vOk AND #iUDT_LiftPI.ix_F1400ok,
	                       ix_SimulationModeActive := "DB_Memory".Simulation,
	                       ix_HardwareOk := #ix_HardwareOk,
	                       qUDT_HMIStatus => #iqUDT_TGWLiftStatus."020".VSU_RIO,
	                       iqUDT_Statistics := #iqUDT_TGWLiftStatistics."020".VSU_RIO,
	                       iqUDT_VSUInterface := #sUDT_020VSUInterface);

	    END_REGION

	    REGION Lift control

	        // add BoS and EoS PEC to this block

	        #sFB_020Lift(iUDT_LiftConveyorInterface := #sUDT_010ConveyorInterface,
	                     iUDT_VSUInterface := #sUDT_020VSUInterface,
	                     ix_SectionIsDown := #sUDT_020VSUInterface.PositionActual = #ci_LiftDown,
	                     ix_SectionIsUp := #sUDT_020VSUInterface.PositionActual = #ci_LiftUp,
	                     ix_PECLift := #ix_010PECMiddle,
	                     ix_ConveyorEmptyInAuto := #iqUDT_InfeedEmptyUpCommonStatus.AutoON,             // Infeed UP
	                     ix_ConveyorEmptyOutAuto := #iqUDT_OutfeedEmptyDownCommonStatus.AutoON,             // Outfeed Down
	                     ix_ConveyorFullInAuto := #iqUDT_InfeedFullDownCommonStatus.AutoON,             // Infeed DOWN
	                     ix_ConveyorFullOutAuto := #iqUDT_OutfeedFullupCommonStatus.AutoON,             // Outfeed UP
	                     qi_RequestedPosition => #sUDT_020VSUInterface.RequestedPosition,
	                     qx_TransportIdle => #sFB_020Lift.qx_TransportIdle,
	                     qx_LiftConveyorDirection => #tx_LiftConveyorDirection,
	                     iqUDT_LiftConveyorHandShakeUpstream := #sUDT_010HandshakeUp,
	                     iqUDT_LiftConveyorHandShake := #sUDT_010Handshake,
	                     iqUDT_InfeedEmptyUpHandShake := #iqUDT_InfeedEmptyUpHandShake,
	                     iqUDT_OutfeedEmptyDownHandShake := #iqUDT_OutfeedEmptyDownHandShake,
	                     iqUDT_InfeedFullDownHandShake := #iqUDT_InfeedFullDownHandShake,
	                     iqUDT_OutfeedFullUpHandShake := #iqUDT_OutfeedFullUpHandShake,
	                     iqUDT_OutfeedFullUpHandshakeUpstream := #iqUDT_OutfeedFullUpHandshakeUpstream,
	                     iqUDT_OutfeedEmptyDownHandshakeUpstream := #iqUDT_OutfeedEmptyDownHandshakeUpstream);

	    END_REGION

	    REGION VSU

	        // add the EoS and BoS to the lift Status, remove from conveyor. Lift block will check the PEC and control the conveyor accordingly

	        #sFB_020VSULift(iUDT_VSUConfig := #iUDT_TGWLiftConfiguration."020".VSU,
	                        ix_SafetyOk := #ix_SafetyOk,
	                        ix_BeltTear1 := #iUDT_LiftPI.ix_BeltTearLeft,
	                        ix_BeltTear2 := #iUDT_LiftPI.ix_BeltTearRight,
	                        ix_MaintSupport1 := #ix_MaintSupport1,
	                        ix_MaintSupport2 := #ix_MaintSupport2,
	                        ix_PosUp := #sUDT_020VSUInterface.PositionActual = #ci_LiftUp,
	                        ix_PosDown := #sUDT_020VSUInterface.PositionActual = #ci_LiftDown,
	                        ix_PECGapEnd := #ix_010PECGapEnd,
	                        ix_PECGapBegin := #ix_010PECGapBegin,
	                        ix_LimitSwitchUp := #ix_LimitSwitchUp,
	                        ix_LimitSwitchDown := #ix_LimitSwitchDown,
	                        ix_SafetyDoorDiagDown := #iUDT_LiftPI.ix_SafetyDoorDownDiag,
	                        ix_SafetyDoorDiagUp := #iUDT_LiftPI.ix_SafetyDoorUpDiag,
	                        ix_LCPAutoMode := #iUDT_LiftPI.ix_AutoMode,
	                        ix_LCPManualMode := #iUDT_LiftPI.ix_ManualMode,
	                        ix_LCPStop := #ix_KeySwitchStop,
	                        ix_LCPDown := #iUDT_LiftPI.ix_JogDown,
	                        ix_LCPUp := #iUDT_LiftPI.ix_JogUp,
	                        ix_LCPRef := #iUDT_LiftPI.ix_Reference,
	                        ix_TransportIdle := #sFB_020Lift.qx_TransportIdle,
	                        ix_HardwareOk := #ix_HardwareOk,
	                        ix_MaintenanceSwitchUp := #iUDT_LiftPI.ix_MaintenanceSwitchUpOn,
	                        ix_MainContactorFeedback := #iUDT_LiftPI.ix_MainContactorFeedbackOn,
	                        ix_OverTempBrakingResistor := #iUDT_LiftPI.ix_OverTempBrakeRes,
	                        qUDT_HMIStatus => #iqUDT_TGWLiftStatus."020".VSU,
	                        qUDT_Status => #iqUDT_TGWLiftCommonStatus."020",
	                        qx_MainContactorOn => #qUDT_LiftPO.qx_MainContactorOn,
	                        iqUDT_EquipmentControl := #iqUDT_EquipmentControl,
	                        iqUDT_VSUCommand := #iqUDT_TGWLiftHMICommands."020".VSU,
	                        iqUDT_VSUInterface := #sUDT_020VSUInterface,
	                        iqUDT_Statistics := #iqUDT_TGWLiftStatistics."020".VSU);

	    END_REGION

	    REGION SEW VFD MOVI-C Positioning

	        #"sFB_020VfdSEWMOVICPositioning"(iUDT_VfdConfig := #iUDT_TGWLiftConfiguration."020".VFD,
	                                         iUDT_VfdInputs := #iUDT_020MotorInput,
	                                         ix_MainPowerOk := TRUE,
	                                         ix_BackupPowerOk := TRUE,
	                                         ix_SimulationModeActive := "DB_Memory".Simulation,
	                                         qUDT_HMIStatus => #iqUDT_TGWLiftStatus."020".VFD,
	                                         qUDT_VfdOutputs => #qUDT_020MotorOutput,
	                                         iqUDT_VSUInterface := #sUDT_020VSUInterface,
	                                         iqUDT_VFDStatistics := #iqUDT_TGWLiftStatistics."020".VFD);

	    END_REGION

	    REGION Signaling
	        // Fault lamp
	        #qUDT_LiftPO.qx_Fault :=
	        #iqUDT_TGWLiftCommonStatus."010".Error
	        OR #iqUDT_TGWLiftCommonStatus."010".SafetyStop
	        OR #iqUDT_TGWLiftCommonStatus."020".Error
	        OR #iqUDT_TGWLiftCommonStatus."020".SafetyStop
	        OR #iqUDT_InfeedEmptyUpCommonStatus.Error
	        OR #iqUDT_InfeedEmptyUpCommonStatus.SafetyStop
	        OR #iqUDT_InfeedFullDownCommonStatus.Error
	        OR #iqUDT_InfeedFullDownCommonStatus.SafetyStop
	        OR #iqUDT_OutfeedEmptyDownCommonStatus.Error
	        OR #iqUDT_OutfeedEmptyDownCommonStatus.SafetyStop
	        OR #iqUDT_OutfeedFullupCommonStatus.Error
	        OR #iqUDT_OutfeedFullupCommonStatus.SafetyStop
	        ;

	    END_REGION

	END_REGION
END_FUNCTION_BLOCK

FUNCTION_BLOCK "FB_WSL"
{ S7_Optimized_Access := 'TRUE' }
VERSION : 0.1
// ATTRIBUTES
// AUTO_NUMBER = True
// BLOCK_NUMBER = 264
// END_ATTRIBUTES
   VAR_INPUT
      iUDT_Configuration { ExternalAccessible := 'False'; ExternalVisible := 'False'; ExternalWritable := 'False'} : "UDT_WSLConfiguration";   // Workstation configuration structure
      iUDT_MotorInput010 { ExternalAccessible := 'False'; ExternalVisible := 'False'; ExternalWritable := 'False'} : "UDT_AixPlcFullIn";   // 010 ConveyLinxAix inputs structure
      iUDT_MotorInput030 { ExternalAccessible := 'False'; ExternalVisible := 'False'; ExternalWritable := 'False'} : "UDT_AixPlcFullIn";   // 030 ConveyLinxAix inputs structure
      iUDT_MotorInput040 { ExternalAccessible := 'False'; ExternalVisible := 'False'; ExternalWritable := 'False'} : "UDT_AixPlcFullIn";   // 030 ConveyLinxAix inputs structure
      iUDT_MotorInput050 { ExternalAccessible := 'False'; ExternalVisible := 'False'; ExternalWritable := 'False'} : "UDT_AixPlcFullIn";   // 050 ConveyLinxAix inputs structure
      iUDT_MotorInput060 { ExternalAccessible := 'False'; ExternalVisible := 'False'; ExternalWritable := 'False'} : "UDT_AixPlcFullIn";   // 060 ConveyLinxAix inputs structure
      iUDT_MotorInput070 { ExternalAccessible := 'False'; ExternalVisible := 'False'; ExternalWritable := 'False'} : "UDT_AixPlcFullIn";   // 070 ConveyLinxAix inputs structure
      iUDT_MotorInput080 { ExternalAccessible := 'False'; ExternalVisible := 'False'; ExternalWritable := 'False'} : "UDT_AixPlcFullIn";   // 080 ConveyLinxAix inputs structure
      iUDT_MotorInput090 { ExternalAccessible := 'False'; ExternalVisible := 'False'; ExternalWritable := 'False'} : "UDT_AixPlcFullIn";   // 090 ConveyLinxAix inputs structure
      iUDT_MotorInput100 { ExternalAccessible := 'False'; ExternalVisible := 'False'; ExternalWritable := 'False'} : "UDT_AixPlcFullIn";   // 100 ConveyLinxAix inputs structure
      iUDT_MotorInput110 { ExternalAccessible := 'False'; ExternalVisible := 'False'; ExternalWritable := 'False'} : "UDT_AixPlcFullIn";   // 110 ConveyLinxAix inputs structure
      iUDT_MotorInput120 { ExternalAccessible := 'False'; ExternalVisible := 'False'; ExternalWritable := 'False'} : "UDT_AixPlcFullIn";   // 120 ConveyLinxAix inputs structure
      iUDT_MotorInput210 { ExternalAccessible := 'False'; ExternalVisible := 'False'; ExternalWritable := 'False'} : "UDT_AixPlcFullIn";   // 210 ConveyLinxAix inputs structure
      iUDT_MotorInput220 { ExternalAccessible := 'False'; ExternalVisible := 'False'; ExternalWritable := 'False'} : "UDT_AixPlcFullIn";   // 220 ConveyLinxAix inputs structure
      iUDT_MotorInput230 { ExternalAccessible := 'False'; ExternalVisible := 'False'; ExternalWritable := 'False'} : "UDT_AixPlcFullIn";   // 230 ConveyLinxAix inputs structure
      iUDT_MotorInput240 { ExternalAccessible := 'False'; ExternalVisible := 'False'; ExternalWritable := 'False'} : "UDT_AixPlcFullIn";   // 240 ConveyLinxAix inputs structure
      iUDT_MotorInput250 { ExternalAccessible := 'False'; ExternalVisible := 'False'; ExternalWritable := 'False'} : "UDT_AixPlcFullIn";   // 250 ConveyLinxAix inputs structure
      iUDT_MotorInput260 { ExternalAccessible := 'False'; ExternalVisible := 'False'; ExternalWritable := 'False'} : "UDT_AixPlcFullIn";   // 260 ConveyLinxAix inputs structure
      iUDT_MotorInput270 { ExternalAccessible := 'False'; ExternalVisible := 'False'; ExternalWritable := 'False'} : "UDT_AixPlcFullIn";   // 270 ConveyLinxAix inputs structure
      iUDT_MotorInput280 { ExternalAccessible := 'False'; ExternalVisible := 'False'; ExternalWritable := 'False'} : "UDT_AixPlcFullIn";   // 280 ConveyLinxAix inputs structure
      iUDT_MotorInput290 { ExternalAccessible := 'False'; ExternalVisible := 'False'; ExternalWritable := 'False'} : "UDT_AixPlcFullIn";   // 290 ConveyLinxAix inputs structure
      iUDT_MotorInput300 { ExternalAccessible := 'False'; ExternalVisible := 'False'; ExternalWritable := 'False'} : "UDT_AixPlcFullIn";   // 300 ConveyLinxAix inputs structure
      iUDT_MotorInput410 { ExternalAccessible := 'False'; ExternalVisible := 'False'; ExternalWritable := 'False'} : "UDT_AixPlcFullIn";   // 410 ConveyLinxAix inputs structure
      iUDT_MotorInput420 { ExternalAccessible := 'False'; ExternalVisible := 'False'; ExternalWritable := 'False'} : "UDT_AixPlcFullIn";   // 420 ConveyLinxAix inputs structure
      iUDT_MotorInput430 { ExternalAccessible := 'False'; ExternalVisible := 'False'; ExternalWritable := 'False'} : "UDT_AixPlcFullIn";   // 430 ConveyLinxAix inputs structure
      iUDT_MotorInput440 { ExternalAccessible := 'False'; ExternalVisible := 'False'; ExternalWritable := 'False'} : "UDT_AixPlcFullIn";   // 440 ConveyLinxAix inputs structure
      iUDT_MotorInput450 { ExternalAccessible := 'False'; ExternalVisible := 'False'; ExternalWritable := 'False'} : "UDT_AixPlcFullIn";   // 450 ConveyLinxAix inputs structure
      iUDT_MotorInput460 { ExternalAccessible := 'False'; ExternalVisible := 'False'; ExternalWritable := 'False'} : "UDT_AixPlcFullIn";   // 460 ConveyLinxAix inputs structure
      iUDT_MotorInput470 { ExternalAccessible := 'False'; ExternalVisible := 'False'; ExternalWritable := 'False'} : "UDT_AixPlcFullIn";   // 470 ConveyLinxAix inputs structure
      iUDT_MotorInput480 { ExternalAccessible := 'False'; ExternalVisible := 'False'; ExternalWritable := 'False'} : "UDT_AixPlcFullIn";   // 480 ConveyLinxAix inputs structure
      iUDT_MotorInput490 { ExternalAccessible := 'False'; ExternalVisible := 'False'; ExternalWritable := 'False'} : "UDT_AixPlcFullIn";   // 490 ConveyLinxAix inputs structure
      iUDT_MotorInput500 { ExternalAccessible := 'False'; ExternalVisible := 'False'; ExternalWritable := 'False'} : "UDT_AixPlcFullIn";   // 500 ConveyLinxAix inputs structure
      iUDT_MotorInput610 { ExternalAccessible := 'False'; ExternalVisible := 'False'; ExternalWritable := 'False'} : "UDT_AixPlcFullIn";   // 610 ConveyLinxAix inputs structure
      iUDT_MotorInput620 { ExternalAccessible := 'False'; ExternalVisible := 'False'; ExternalWritable := 'False'} : "UDT_AixPlcFullIn";   // 620 ConveyLinxAix inputs structure
      iUDT_MotorInput630 { ExternalAccessible := 'False'; ExternalVisible := 'False'; ExternalWritable := 'False'} : "UDT_AixPlcFullIn";   // 630 ConveyLinxAix inputs structure
      iUDT_MotorInput640 { ExternalAccessible := 'False'; ExternalVisible := 'False'; ExternalWritable := 'False'} : "UDT_AixPlcFullIn";   // 640 ConveyLinxAix inputs structure
      iUDT_ScannerInput280 { ExternalAccessible := 'False'; ExternalVisible := 'False'; ExternalWritable := 'False'} : "UDT_CognexDM260_IN";   // Cognex inputs structur
      iUDT_ScannerInput480 { ExternalAccessible := 'False'; ExternalVisible := 'False'; ExternalWritable := 'False'} : "UDT_CognexDM260_IN";
      ix_24vOk { ExternalAccessible := 'False'; ExternalVisible := 'False'; ExternalWritable := 'False'} : Bool;   // TRUE when 24VDC is healthy
      ix_400vOk { ExternalAccessible := 'False'; ExternalVisible := 'False'; ExternalWritable := 'False'} : Bool;   // TRUE when 400VAC is healthy
      ix_SafetyOk { ExternalAccessible := 'False'; ExternalVisible := 'False'; ExternalWritable := 'False'} : Bool;   // TRUE when safety is ok
      ix_HardwareOk { ExternalAccessible := 'False'; ExternalVisible := 'False'; ExternalWritable := 'False'} : Bool;   // TRUE when hardware is ok
      ix_AirPressureOk { ExternalAccessible := 'False'; ExternalVisible := 'False'; ExternalWritable := 'False'} : Bool;   // TRUE when air pressure is ok
      ix_SectionIsUp121 { ExternalAccessible := 'False'; ExternalVisible := 'False'; ExternalWritable := 'False'} : Bool;   // TRUE when section 121 is up
      ix_SectionIsDown121 { ExternalAccessible := 'False'; ExternalVisible := 'False'; ExternalWritable := 'False'} : Bool;   // TRUE when section 121 is down
      ix_SectionIsUp221 { ExternalAccessible := 'False'; ExternalVisible := 'False'; ExternalWritable := 'False'} : Bool;   // TRUE when section 221  is up
      ix_SectionIsDown221 { ExternalAccessible := 'False'; ExternalVisible := 'False'; ExternalWritable := 'False'} : Bool;   // TRUE when section 221 is down
      ix_SectionIsUp291 { ExternalAccessible := 'False'; ExternalVisible := 'False'; ExternalWritable := 'False'} : Bool;   // TRUE when section 291 is up
      ix_SectionIsDown291 { ExternalAccessible := 'False'; ExternalVisible := 'False'; ExternalWritable := 'False'} : Bool;   // TRUE when section 291 is down
      ix_SectionIsUp421 { ExternalAccessible := 'False'; ExternalVisible := 'False'; ExternalWritable := 'False'} : Bool;   // TRUE when section 421 is up
      ix_SectionIsDown421 { ExternalAccessible := 'False'; ExternalVisible := 'False'; ExternalWritable := 'False'} : Bool;   // TRUE when section 421 is down
      ix_SectionIsUp491 { ExternalAccessible := 'False'; ExternalVisible := 'False'; ExternalWritable := 'False'} : Bool;   // TRUE when section 491 is up
      ix_SectionIsDown491 { ExternalAccessible := 'False'; ExternalVisible := 'False'; ExternalWritable := 'False'} : Bool;   // TRUE when section 491 is down
      ix_SectionIsUp611 { ExternalAccessible := 'False'; ExternalVisible := 'False'; ExternalWritable := 'False'} : Bool;   // TRUE when section 611 is up
      ix_SectionIsDown611 { ExternalAccessible := 'False'; ExternalVisible := 'False'; ExternalWritable := 'False'} : Bool;   // TRUE when section 611 is down
      ix_Done490 { ExternalAccessible := 'False'; ExternalVisible := 'False'; ExternalWritable := 'False'} : Bool;   // TRUE if action on right station is done and bin is ready to be send away
      ix_Done290 { ExternalAccessible := 'False'; ExternalVisible := 'False'; ExternalWritable := 'False'} : Bool;   // TRUE if action on left station is done and bin is ready to be send away
   END_VAR

   VAR_OUTPUT
      qUDT_MotorOutput010 { ExternalAccessible := 'False'; ExternalVisible := 'False'; ExternalWritable := 'False'} : "UDT_AixPlcFullOut";   // 010 ConveyLinxAix outputs structure
      qUDT_MotorOutput030 { ExternalAccessible := 'False'; ExternalVisible := 'False'; ExternalWritable := 'False'} : "UDT_AixPlcFullOut";   // 030 ConveyLinxAix outputs structure
      qUDT_MotorOutput040 { ExternalAccessible := 'False'; ExternalVisible := 'False'; ExternalWritable := 'False'} : "UDT_AixPlcFullOut";   // 040 ConveyLinxAix outputs structure
      qUDT_MotorOutput050 { ExternalAccessible := 'False'; ExternalVisible := 'False'; ExternalWritable := 'False'} : "UDT_AixPlcFullOut";   // 050 ConveyLinxAix outputs structure
      qUDT_MotorOutput060 { ExternalAccessible := 'False'; ExternalVisible := 'False'; ExternalWritable := 'False'} : "UDT_AixPlcFullOut";   // 060 ConveyLinxAix outputs structure
      qUDT_MotorOutput070 { ExternalAccessible := 'False'; ExternalVisible := 'False'; ExternalWritable := 'False'} : "UDT_AixPlcFullOut";   // 070 ConveyLinxAix outputs structure
      qUDT_MotorOutput080 { ExternalAccessible := 'False'; ExternalVisible := 'False'; ExternalWritable := 'False'} : "UDT_AixPlcFullOut";   // 080 ConveyLinxAix outputs structure
      qUDT_MotorOutput090 { ExternalAccessible := 'False'; ExternalVisible := 'False'; ExternalWritable := 'False'} : "UDT_AixPlcFullOut";   // 090 ConveyLinxAix outputs structure
      qUDT_MotorOutput100 { ExternalAccessible := 'False'; ExternalVisible := 'False'; ExternalWritable := 'False'} : "UDT_AixPlcFullOut";   // 100 ConveyLinxAix outputs structure
      qUDT_MotorOutput110 { ExternalAccessible := 'False'; ExternalVisible := 'False'; ExternalWritable := 'False'} : "UDT_AixPlcFullOut";   // 110 ConveyLinxAix outputs structure
      qUDT_MotorOutput120 { ExternalAccessible := 'False'; ExternalVisible := 'False'; ExternalWritable := 'False'} : "UDT_AixPlcFullOut";   // 120 ConveyLinxAix outputs structure
      qUDT_MotorOutput210 { ExternalAccessible := 'False'; ExternalVisible := 'False'; ExternalWritable := 'False'} : "UDT_AixPlcFullOut";   // 210 ConveyLinxAix outputs structure
      qUDT_MotorOutput220 { ExternalAccessible := 'False'; ExternalVisible := 'False'; ExternalWritable := 'False'} : "UDT_AixPlcFullOut";   // 220 ConveyLinxAix outputs structure
      qUDT_MotorOutput230 { ExternalAccessible := 'False'; ExternalVisible := 'False'; ExternalWritable := 'False'} : "UDT_AixPlcFullOut";   // 230 ConveyLinxAix outputs structure
      qUDT_MotorOutput240 { ExternalAccessible := 'False'; ExternalVisible := 'False'; ExternalWritable := 'False'} : "UDT_AixPlcFullOut";   // 240 ConveyLinxAix outputs structure
      qUDT_MotorOutput250 { ExternalAccessible := 'False'; ExternalVisible := 'False'; ExternalWritable := 'False'} : "UDT_AixPlcFullOut";   // 250 ConveyLinxAix outputs structure
      qUDT_MotorOutput260 { ExternalAccessible := 'False'; ExternalVisible := 'False'; ExternalWritable := 'False'} : "UDT_AixPlcFullOut";   // 260 ConveyLinxAix outputs structure
      qUDT_MotorOutput270 { ExternalAccessible := 'False'; ExternalVisible := 'False'; ExternalWritable := 'False'} : "UDT_AixPlcFullOut";   // 270 ConveyLinxAix outputs structure
      qUDT_MotorOutput280 { ExternalAccessible := 'False'; ExternalVisible := 'False'; ExternalWritable := 'False'} : "UDT_AixPlcFullOut";   // 280 ConveyLinxAix outputs structure
      qUDT_MotorOutput290 { ExternalAccessible := 'False'; ExternalVisible := 'False'; ExternalWritable := 'False'} : "UDT_AixPlcFullOut";   // 290 ConveyLinxAix outputs structure
      qUDT_MotorOutput300 { ExternalAccessible := 'False'; ExternalVisible := 'False'; ExternalWritable := 'False'} : "UDT_AixPlcFullOut";   // 300 ConveyLinxAix outputs structure
      qUDT_MotorOutput410 { ExternalAccessible := 'False'; ExternalVisible := 'False'; ExternalWritable := 'False'} : "UDT_AixPlcFullOut";   // 410 ConveyLinxAix outputs structure
      qUDT_MotorOutput420 { ExternalAccessible := 'False'; ExternalVisible := 'False'; ExternalWritable := 'False'} : "UDT_AixPlcFullOut";   // 420 ConveyLinxAix outputs structure
      qUDT_MotorOutput430 { ExternalAccessible := 'False'; ExternalVisible := 'False'; ExternalWritable := 'False'} : "UDT_AixPlcFullOut";   // 430 ConveyLinxAix outputs structure
      qUDT_MotorOutput440 { ExternalAccessible := 'False'; ExternalVisible := 'False'; ExternalWritable := 'False'} : "UDT_AixPlcFullOut";   // 440 ConveyLinxAix outputs structure
      qUDT_MotorOutput450 { ExternalAccessible := 'False'; ExternalVisible := 'False'; ExternalWritable := 'False'} : "UDT_AixPlcFullOut";   // 450 ConveyLinxAix outputs structure
      qUDT_MotorOutput460 { ExternalAccessible := 'False'; ExternalVisible := 'False'; ExternalWritable := 'False'} : "UDT_AixPlcFullOut";   // 460 ConveyLinxAix outputs structure
      qUDT_MotorOutput470 { ExternalAccessible := 'False'; ExternalVisible := 'False'; ExternalWritable := 'False'} : "UDT_AixPlcFullOut";   // 470 ConveyLinxAix outputs structure
      qUDT_MotorOutput480 { ExternalAccessible := 'False'; ExternalVisible := 'False'; ExternalWritable := 'False'} : "UDT_AixPlcFullOut";   // 480 ConveyLinxAix outputs structure
      qUDT_MotorOutput490 { ExternalAccessible := 'False'; ExternalVisible := 'False'; ExternalWritable := 'False'} : "UDT_AixPlcFullOut";   // 490 ConveyLinxAix outputs structure
      qUDT_MotorOutput500 { ExternalAccessible := 'False'; ExternalVisible := 'False'; ExternalWritable := 'False'} : "UDT_AixPlcFullOut";   // 500 ConveyLinxAix outputs structure
      qUDT_MotorOutput610 { ExternalAccessible := 'False'; ExternalVisible := 'False'; ExternalWritable := 'False'} : "UDT_AixPlcFullOut";   // 610 ConveyLinxAix outputs structure
      qUDT_MotorOutput620 { ExternalAccessible := 'False'; ExternalVisible := 'False'; ExternalWritable := 'False'} : "UDT_AixPlcFullOut";   // 620 ConveyLinxAix outputs structure
      qUDT_MotorOutput630 { ExternalAccessible := 'False'; ExternalVisible := 'False'; ExternalWritable := 'False'} : "UDT_AixPlcFullOut";   // 630 ConveyLinxAix outputs structure
      qUDT_MotorOutput640 { ExternalAccessible := 'False'; ExternalVisible := 'False'; ExternalWritable := 'False'} : "UDT_AixPlcFullOut";   // 640 ConveyLinxAix outputs structure
      qUDT_ScannerOutput280 { ExternalAccessible := 'False'; ExternalVisible := 'False'; ExternalWritable := 'False'} : "UDT_CognexDM260_OUT";   // Cognex output structure
      qUDT_ScannerOutput480 { ExternalAccessible := 'False'; ExternalVisible := 'False'; ExternalWritable := 'False'} : "UDT_CognexDM260_OUT";
      qx_PopupControl121 { ExternalAccessible := 'False'; ExternalVisible := 'False'; ExternalWritable := 'False'} : Bool;   // Command up for section 121
      qx_PopupControl221 { ExternalAccessible := 'False'; ExternalVisible := 'False'; ExternalWritable := 'False'} : Bool;   // Command up for section 221
      qx_PopupControl291 { ExternalAccessible := 'False'; ExternalVisible := 'False'; ExternalWritable := 'False'} : Bool;   // Command up for section 291
      qx_PopupControl421 { ExternalAccessible := 'False'; ExternalVisible := 'False'; ExternalWritable := 'False'} : Bool;   // Command up for section 421
      qx_PopupControl491 { ExternalAccessible := 'False'; ExternalVisible := 'False'; ExternalWritable := 'False'} : Bool;   // Command up for section 491
      qx_PopupControl611 { ExternalAccessible := 'False'; ExternalVisible := 'False'; ExternalWritable := 'False'} : Bool;   // Command up for section 611
   END_VAR

   VAR_IN_OUT
      iqUDT_EquipmentControl : "UDT_EquipmentControl";   // Equipment control structure
      iqUDT_HandshakeUpstream010 : "UDT_ConveyorHandshake";   // Upstream handshake structure for 010 conveyor
      iqUDT_HandshakeDownstream640 : "UDT_ConveyorHandshake";   // Downstream handshake structure for 640 conveyor
      iqUDT_WorkstationCommands : "UDT_WSLHmiCommands";   // Workstation command structure
      iqUDT_WorkstationStatistics : "UDT_WSLStatistics";   // Statistics structure
      iqUDT_WorkstationStatus : "UDT_WSLStatus";   // HMI Status structure
      iqUDT_WorkstationCommonStatus : "UDT_WSLCommonStatus";   // Common status structure
      iqUDT_RATPositioning120 : "UDT_RATPositioning";   // Structure including data for servo control RAT 121
      iqUDT_RATPositioning220 : "UDT_RATPositioning";   // Structure including data for servo control RAT 221
      iqUDT_RATPositioning290 : "UDT_RATPositioning";   // Structure including data for servo control RAT 291
      iqUDT_RATPositioning420 : "UDT_RATPositioning";   // Structure including data for servo control RAT 421
      iqUDT_RATPositioning490 : "UDT_RATPositioning";   // Structure including data for servo control RAT 491
      iqUDT_RATPositioning610 : "UDT_RATPositioning";   // Structure including data for servo control RAT 611
   END_VAR

